{attribute 'GeneratedUsingTerminal: EK1960-0000-0019'}
{attribute addProperty BoxType "EK1960-0000-0019"}
{attribute addProperty Id "FSoE_CommandUSINT1FSOUT_Module_1_Channel_1_OutputBOOL1FSOUT_Module_1_Channel_2_OutputBOOL1FSOUT_Module_1_Channel_3_OutputBOOL1FSOUT_Module_1_Channel_4_OutputBOOL1FSOUT_Module_1_ErrAckBOOL1FSOUT_Module_2_Channel_1_OutputBOOL1FSOUT_Module_2_Channel_2_OutputBOOL1FSOUT_Module_2_Channel_3_OutputBOOL1FSOUT_Module_2_Channel_4_OutputBOOL1FSOUT_Module_2_ErrAckBOOL1FSOUT_Module_3_Channel_1_OutputBOOL1FSOUT_Module_3_Channel_2_OutputBOOL1FSOUT_Module_3_Channel_3_OutputBOOL1FSOUT_Module_3_Channel_4_OutputBOOL1FSOUT_Module_3_ErrAckBOOL1FSOUT_Module_4_Channel_1_OutputBOOL1FSoE_CRC_000UINT2FSOUT_Module_4_Channel_2_OutputBOOL1FSOUT_Module_4_Channel_3_OutputBOOL1FSOUT_Module_4_Channel_4_OutputBOOL1FSOUT_Module_4_ErrAckBOOL1FSOUT_Module_5_Channel_1_OutputBOOL1FSOUT_Module_5_Channel_2_OutputBOOL1FSOUT_Module_5_Channel_3_OutputBOOL1FSOUT_Module_5_Channel_4_OutputBOOL1FSOUT_Module_5_ErrAckBOOL1FSOUT_Module_6_Channel_1_OutputBOOL1FSOUT_Module_6_Channel_2_OutputBOOL1FSOUT_Module_6_Channel_3_OutputBOOL1FSOUT_Module_6_Channel_4_OutputBOOL1FSOUT_Module_6_ErrAckBOOL1FSoE_CRC_001UINT2FSIN_Module_1_ErrAckBOOL1FSIN_Module_2_ErrAckBOOL1FSIN_Module_3_ErrAckBOOL1FSIN_Module_4_ErrAckBOOL1FSIN_Module_5_ErrAckBOOL1FSIN_Module_6_ErrAckBOOL1FSIN_Module_7_ErrAckBOOL1FSIN_Module_8_ErrAckBOOL1FSIN_Module_9_ErrAck_1BOOL1FSIN_Module_9_ErrAck_2BOOL1FSIN_Module_10_ErrAck_1BOOL1FSIN_Module_10_ErrAck_2BOOL1FSoE_CRC_002UINT2FSoE_Connection_IDUINT2"}
{attribute addProperty CRC "3133652769"}
{attribute addProperty Size "51"}
TYPE FSOE_BAC7BF21 :
STRUCT
	{attribute addProperty Name "FSoE_Command"}
	FSoE_Command : USINT;
	{attribute addProperty Name "FSOUT_Module_1_Channel_1_Output"}
	FSOUT_Module_1_Channel_1_Output : BOOL;
	{attribute addProperty Name "FSOUT_Module_1_Channel_2_Output"}
	FSOUT_Module_1_Channel_2_Output : BOOL;
	{attribute addProperty Name "FSOUT_Module_1_Channel_3_Output"}
	FSOUT_Module_1_Channel_3_Output : BOOL;
	{attribute addProperty Name "FSOUT_Module_1_Channel_4_Output"}
	FSOUT_Module_1_Channel_4_Output : BOOL;
	{attribute addProperty Name "FSOUT_Module_1_ErrAck"}
	FSOUT_Module_1_ErrAck : BOOL;
	{attribute addProperty Name "FSOUT_Module_2_Channel_1_Output"}
	FSOUT_Module_2_Channel_1_Output : BOOL;
	{attribute addProperty Name "FSOUT_Module_2_Channel_2_Output"}
	FSOUT_Module_2_Channel_2_Output : BOOL;
	{attribute addProperty Name "FSOUT_Module_2_Channel_3_Output"}
	FSOUT_Module_2_Channel_3_Output : BOOL;
	{attribute addProperty Name "FSOUT_Module_2_Channel_4_Output"}
	FSOUT_Module_2_Channel_4_Output : BOOL;
	{attribute addProperty Name "FSOUT_Module_2_ErrAck"}
	FSOUT_Module_2_ErrAck : BOOL;
	{attribute addProperty Name "FSOUT_Module_3_Channel_1_Output"}
	FSOUT_Module_3_Channel_1_Output : BOOL;
	{attribute addProperty Name "FSOUT_Module_3_Channel_2_Output"}
	FSOUT_Module_3_Channel_2_Output : BOOL;
	{attribute addProperty Name "FSOUT_Module_3_Channel_3_Output"}
	FSOUT_Module_3_Channel_3_Output : BOOL;
	{attribute addProperty Name "FSOUT_Module_3_Channel_4_Output"}
	FSOUT_Module_3_Channel_4_Output : BOOL;
	{attribute addProperty Name "FSOUT_Module_3_ErrAck"}
	FSOUT_Module_3_ErrAck : BOOL;
	{attribute addProperty Name "FSOUT_Module_4_Channel_1_Output"}
	FSOUT_Module_4_Channel_1_Output : BOOL;
	{attribute addProperty Name "FSoE_CRC_000"}
	FSoE_CRC_000 : UINT;
	{attribute addProperty Name "FSOUT_Module_4_Channel_2_Output"}
	FSOUT_Module_4_Channel_2_Output : BOOL;
	{attribute addProperty Name "FSOUT_Module_4_Channel_3_Output"}
	FSOUT_Module_4_Channel_3_Output : BOOL;
	{attribute addProperty Name "FSOUT_Module_4_Channel_4_Output"}
	FSOUT_Module_4_Channel_4_Output : BOOL;
	{attribute addProperty Name "FSOUT_Module_4_ErrAck"}
	FSOUT_Module_4_ErrAck : BOOL;
	{attribute addProperty Name "FSOUT_Module_5_Channel_1_Output"}
	FSOUT_Module_5_Channel_1_Output : BOOL;
	{attribute addProperty Name "FSOUT_Module_5_Channel_2_Output"}
	FSOUT_Module_5_Channel_2_Output : BOOL;
	{attribute addProperty Name "FSOUT_Module_5_Channel_3_Output"}
	FSOUT_Module_5_Channel_3_Output : BOOL;
	{attribute addProperty Name "FSOUT_Module_5_Channel_4_Output"}
	FSOUT_Module_5_Channel_4_Output : BOOL;
	{attribute addProperty Name "FSOUT_Module_5_ErrAck"}
	FSOUT_Module_5_ErrAck : BOOL;
	{attribute addProperty Name "FSOUT_Module_6_Channel_1_Output"}
	FSOUT_Module_6_Channel_1_Output : BOOL;
	{attribute addProperty Name "FSOUT_Module_6_Channel_2_Output"}
	FSOUT_Module_6_Channel_2_Output : BOOL;
	{attribute addProperty Name "FSOUT_Module_6_Channel_3_Output"}
	FSOUT_Module_6_Channel_3_Output : BOOL;
	{attribute addProperty Name "FSOUT_Module_6_Channel_4_Output"}
	FSOUT_Module_6_Channel_4_Output : BOOL;
	{attribute addProperty Name "FSOUT_Module_6_ErrAck"}
	FSOUT_Module_6_ErrAck : BOOL;
	{attribute addProperty Name "FSoE_CRC_001"}
	FSoE_CRC_001 : UINT;
	{attribute addProperty Name "FSIN_Module_1_ErrAck"}
	FSIN_Module_1_ErrAck : BOOL;
	{attribute addProperty Name "FSIN_Module_2_ErrAck"}
	FSIN_Module_2_ErrAck : BOOL;
	{attribute addProperty Name "FSIN_Module_3_ErrAck"}
	FSIN_Module_3_ErrAck : BOOL;
	{attribute addProperty Name "FSIN_Module_4_ErrAck"}
	FSIN_Module_4_ErrAck : BOOL;
	{attribute addProperty Name "FSIN_Module_5_ErrAck"}
	FSIN_Module_5_ErrAck : BOOL;
	{attribute addProperty Name "FSIN_Module_6_ErrAck"}
	FSIN_Module_6_ErrAck : BOOL;
	{attribute addProperty Name "FSIN_Module_7_ErrAck"}
	FSIN_Module_7_ErrAck : BOOL;
	{attribute addProperty Name "FSIN_Module_8_ErrAck"}
	FSIN_Module_8_ErrAck : BOOL;
	{attribute addProperty Name "FSIN_Module_9_ErrAck_1"}
	FSIN_Module_9_ErrAck_1 : BOOL;
	{attribute addProperty Name "FSIN_Module_9_ErrAck_2"}
	FSIN_Module_9_ErrAck_2 : BOOL;
	{attribute addProperty Name "FSIN_Module_10_ErrAck_1"}
	FSIN_Module_10_ErrAck_1 : BOOL;
	{attribute addProperty Name "FSIN_Module_10_ErrAck_2"}
	FSIN_Module_10_ErrAck_2 : BOOL;
	{attribute addProperty Name "FSoE_CRC_002"}
	FSoE_CRC_002 : UINT;
	{attribute addProperty Name "FSoE_Connection_ID"}
	FSoE_Connection_ID : UINT;
END_STRUCT
END_TYPE

(* stored: Version 1.2.0.0, ProductVersion 3.1.4024.9
   DUT FSOE_BAC7BF21: Id {304c05ac-ebed-47e6-a02e-bf0bb04950d0} *)
